(* PLC project v0.6.04_CycleSemiAuto.project, CODESYS CODESYS V3.5 SP19 Patch 1 *)
(* stored: creationDateTime 2026-08-14T21:46:21.167793, modificationDateTime 2026-08-14T21:46:21.167793 *)

(* ═══════════════════════════════════════════════════════════════ 🎯 ST_HomingChecklist — Diagnostic chronologique de référencement (Dépannage) ─────────────────────────────────────────────────────────────── 🎨 Permet de localiser immédiatement l'étape qui bloque le Homing (M1/M2). ═══════════════════════════════════════════════════════════════ *)
TYPE ST_HomingChecklist : STRUCT
  Step1_ModeAuthorized : BOOL;  (* 1. Pré-requis de mode TRUE = Mode MAINT_N1 ou MAINT_N2 actif ➔ Commutateur Mode IHM : GVL_IHM.Modes *)
  Step2_WinchSelected : BOOL;  (* TRUE = Treuil sélectionné en MAINT_N2 ➔ Bouton IHM : GVL_IHM.Modes.Cmd.TglJoystickMaster / Selection Treuil *)
  Step3_EncoderAvailable : BOOL;  (* 2. Santé Matériel & Bus TRUE = Codeur EtherCAT OK & E/S OK ➔ Si simu : GVL_Simulation.SimWinchActive=1 / SimSafetyActive=1 *)
  HwIn_ContactorsReleased_DI : BOOL;  (* 2bis. Entrées physiques directes HwIn (vérité terrain) Retours contacteurs retombés issus de HwIn.Winch *)
  HwIn_BrakeIsOpen_DI : BOOL;  (* Retour fin de course frein (1 = ouvert) issu de HwIn.Winch *)
  HwIn_TopPositionFree_DI : BOOL;  (* Capteur position haute commun libre (1 = libre) issu de HwIn.Winch *)
  Step4_ContactorsReleased : BOOL;  (* 3. État Physique Machine TRUE = Tous les contacteurs retombés (attendre l'arrêt complet) *)
  Step5_BrakeApplied : BOOL;  (* TRUE = Frein serré (attendre l'arrêt complet) *)
  TopPositionSensorActive : BOOL;  (* 📍 Fin de course haut physique (TRUE = au contact) *)
  BucketIsOpen : BOOL;  (* 🪣 Benne Ouvert (TRUE = Ouvert) ➔ Pour forcer sans codeur : GVL_IHM.M2TreuilBenne.Bucket.Cmd.BtnConfirmOpenPos *)
  AllConditionsMet : BOOL;  (* 4. Séquence & Bilan TRUE = Prêt pour le homing ! ➔ Déclencher : GVL_IHM.M1TreuilRetenue.Cmd.BtnHome (à 8m) ou BtnHomingAtZero (à 0m) *)
  HomingBusy : BOOL;  (* TRUE = Séquence de calage en cours *)
  HomingDone : BOOL;  (* TRUE = Calage réussi *)
  HomingHomed : BOOL;  (* TRUE = Treuil actuellement référencé *)
  HomingSuspect : BOOL;  (* TRUE = Doute redémarrage ➔ Lever le doute via : GVL_IHM.M1TreuilRetenue.Cmd.BtnConfirmCoherence *)
  RejectErrorMask : WORD;  (* 5. Code de rejet exact Bitmask d'erreur FB_Encoder_Homing.ErrorId *)
END_STRUCT;
END_TYPE
